{attribute 'OPC.UA.DA.StructuredType' := '1'}
FUNCTION_BLOCK FB_DualRedundantSensor EXTENDS FB_BaseDevice IMPLEMENTS I_Device, I_Sensor

VAR
	{attribute 'OPC.UA.DA' := '1'}
  	{attribute 'OPC.UA.DA.StructuredType' := '1'}
	fbSensor1: REFERENCE TO I_Sensor;
	{attribute 'OPC.UA.DA' := '1'}
  	{attribute 'OPC.UA.DA.StructuredType' := '1'}
	fbSensor2: REFERENCE TO I_Sensor;
	{attribute 'OPC.UA.DA' := '1'}
	nCurrentValue: REAL;
	
	eSensorType: E_SensorType;
	
	{attribute 'OPC.UA.DA' := '0'} 
	fbSenso1_vals: ARRAY[1..200] OF REAL;  //Arrays to store last 200 samples of sensors, enabling historic analysis
	{attribute 'OPC.UA.DA' := '0'} 
	fbSenso2_vals: ARRAY[1..200] OF REAL;
	
END_VAR

calculate();

METHOD addSensors : BOOL
VAR_INPUT
	
	Sensor1: REFERENCE TO I_Sensor;
	Sensor2: REFERENCE TO I_Sensor;
	
END_VAR

fbSensor1 := Sensor1;
fbSensor2 := Sensor2;
END_METHOD

METHOD calculate : BOOL
VAR_INPUT
END_VAR
//nCurrentValue := ( fbSensor1.getValue() + fbSensor2.getValue() ) / 2.0;  // calculate average of 2 sensors and return
END_METHOD

METHOD checkCorrelation : BOOL
VAR_INPUT
END_VAR
END_METHOD

{warning 'add method implementation '}
METHOD disable : BOOL
END_METHOD

{warning 'add method implementation '}
METHOD enable : BOOL
END_METHOD

{warning 'add method implementation '}
METHOD FB_init : BOOL
VAR_INPUT
	(* if TRUE, the retain variables are initialized (warm start / cold start)*)
	bInitRetains	: BOOL;
	(* if TRUE, the instance afterwards gets moved into the copy code (online change)*)
	bInCopyCode	: BOOL;
	SensorID	: STRING(80);
	SensorDescr	: STRING(255);
	SensorType	: E_SensorType;
	

	
END_VAR
sID := SensorID;
sDescr := SensorDescr;
eSensorType := SensorType;
END_METHOD

{warning 'add method implementation '}
METHOD getType : E_SensorType
END_METHOD

{warning 'add method implementation '}
METHOD getValue : REAL
END_METHOD

{warning 'add method implementation '}
METHOD write : BOOL
END_METHOD

END_FUNCTION_BLOCK

(* stored: Version 1.1.0.1, ProductVersion 3.1.4024.12
   POU FB_DualRedundantSensor: Id {a5c68a1b-a487-4b48-ac1d-4396ce8245c3}, SpecialFunc None
   Method addSensors: Id {b25eb56e-45ff-4588-a0f0-488590343201}
   Method calculate: Id {7ad4c3a6-32f7-44b3-9963-2b10866d254a}
   Method checkCorrelation: Id {ef7218f3-8352-4a9f-809c-839d41e57faf}
   Method disable: Id {8120a105-8dca-42e0-993c-99aade26fc13}
   Method enable: Id {8835bbf1-a6a7-42f3-9e7b-e72453e610d4}
   Method FB_init: Id {21ad96c2-dadb-4aab-9c6d-66a6c1d353d2}
   Method getType: Id {23ba2315-6878-4867-946c-6c4a39bc5ac3}
   Method getValue: Id {ccfd48c3-6284-46d9-a3b4-aa64aca7f967}
   Method write: Id {2f984d04-9bee-4b11-a561-3b8d9dee2f11} *)
